// TIA Portal V18 export
FUNCTION "Room2_Main" : Void   // FC5, LAD
{ S7_Optimized_Access := 'TRUE' }
VERSION : 0.1
// stored: AutoNumber true, IsIECCheckEnabled false, SetENOAutomatically false, UDAEnableTagReadback false
BEGIN

REGION Network 1: 区域搜索
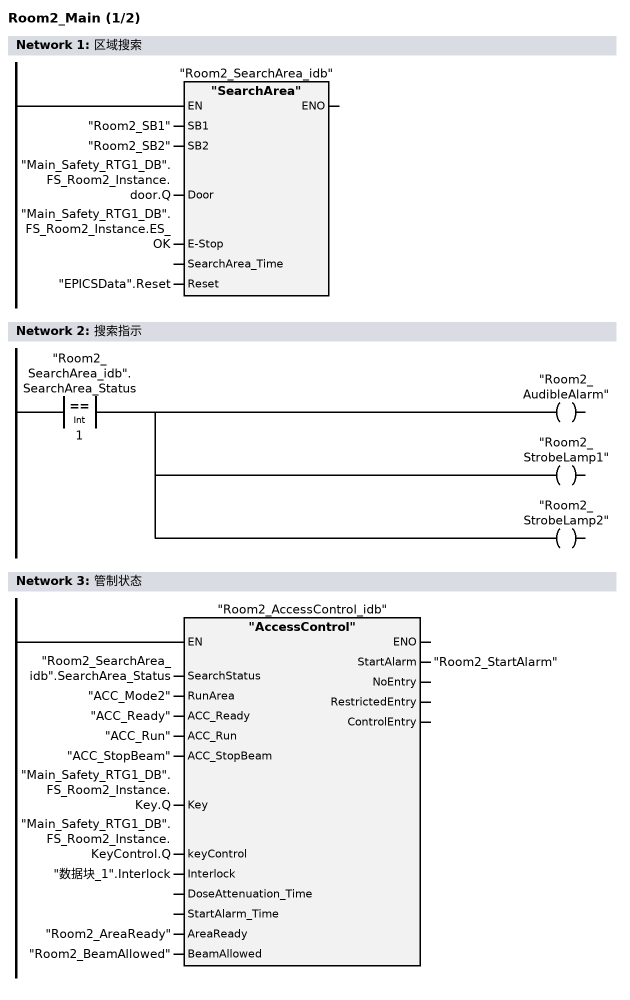
   RUNG wire#powerrail
      "Room2_SearchArea_idb"(SB1 := "Room2_SB1", SB2 := "Room2_SB2", Door := "Main_Safety_RTG1_DB".FS_Room2_Instance.door.Q, "E-Stop" := "Main_Safety_RTG1_DB".FS_Room2_Instance.ES_OK, SearchArea_Time :=, Reset := "EPICSData".Reset)
   END_RUNG
   // the same network as SCL:
   "Room2_SearchArea_idb"(SB1 := "Room2_SB1",   // "SearchArea"
                          SB2 := "Room2_SB2",
                          Door := "Main_Safety_RTG1_DB".FS_Room2_Instance.door.Q,
                          "E-Stop" := "Main_Safety_RTG1_DB".FS_Room2_Instance.ES_OK,
                          Reset := "EPICSData".Reset);
END_REGION

REGION Network 2: 搜索指示
   RUNG wire#powerrail
      { S7_Templates := "SrcType := Int" } EQ_Contact(in1 := "Room2_SearchArea_idb".SearchArea_Status, in2 := 1)
      wire#w1
      Coil( "Room2_AudibleAlarm" )
   END_RUNG
   RUNG wire#w1
      Coil( "Room2_StrobeLamp1" )
   END_RUNG
   RUNG wire#w1
      Coil( "Room2_StrobeLamp2" )
   END_RUNG
   // the same network as SCL:
   "Room2_AudibleAlarm" := "Room2_SearchArea_idb".SearchArea_Status = 1;
   "Room2_StrobeLamp1" := "Room2_AudibleAlarm";
   "Room2_StrobeLamp2" := "Room2_AudibleAlarm";
END_REGION

REGION Network 3: 管制状态
   RUNG wire#powerrail
      "Room2_AccessControl_idb"(SearchStatus := "Room2_SearchArea_idb".SearchArea_Status, RunArea := "ACC_Mode2", ACC_Ready := "ACC_Ready", ACC_Run := "ACC_Run", ACC_StopBeam := "ACC_StopBeam", Key := "Main_Safety_RTG1_DB".FS_Room2_Instance.Key.Q, keyControl := "Main_Safety_RTG1_DB".FS_Room2_Instance.KeyControl.Q, Interlock := "数据块_1".Interlock, DoseAttenuation_Time :=, StartAlarm_Time :=, AreaReady := "Room2_AreaReady", BeamAllowed := "Room2_BeamAllowed", StartAlarm => "Room2_StartAlarm", NoEntry =>, RestrictedEntry =>, ControlEntry =>)
   END_RUNG
   // the same network as SCL:
   "Room2_AccessControl_idb"(SearchStatus := "Room2_SearchArea_idb".SearchArea_Status,   // "AccessControl"
                           RunArea := "ACC_Mode2",
                           ACC_Ready := "ACC_Ready",
                           ACC_Run := "ACC_Run",
                           ACC_StopBeam := "ACC_StopBeam",
                           Key := "Main_Safety_RTG1_DB".FS_Room2_Instance.Key.Q,
                           keyControl := "Main_Safety_RTG1_DB".FS_Room2_Instance.KeyControl.Q,
                           Interlock := "数据块_1".Interlock,
                           AreaReady := "Room2_AreaReady",
                           BeamAllowed := "Room2_BeamAllowed",
                           StartAlarm => "Room2_StartAlarm");
END_REGION

REGION Network 4: 管制输出
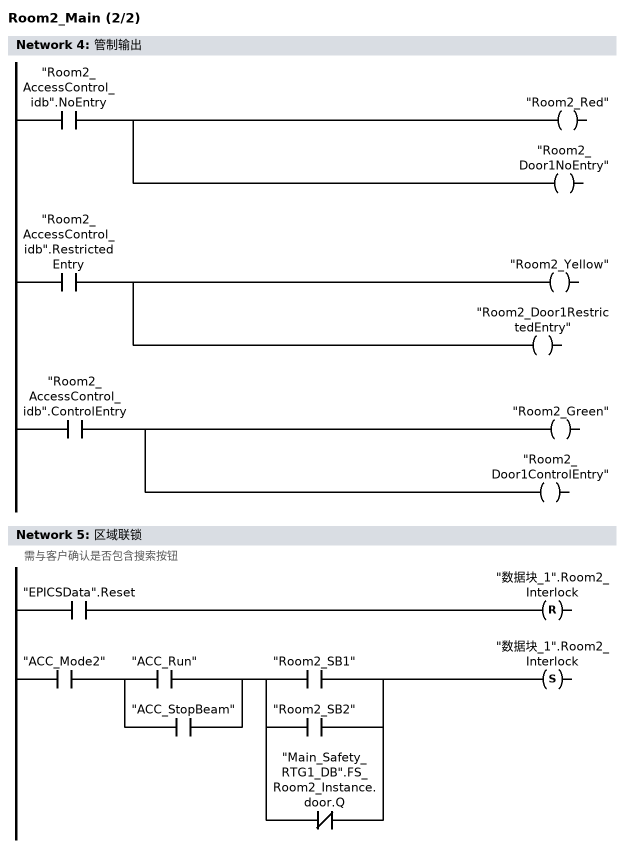
   RUNG wire#powerrail
      Contact( "Room2_AccessControl_idb".NoEntry )
      wire#w1
      Coil( "Room2_Red" )
   END_RUNG
   RUNG wire#w1
      Coil( "Room2_Door1NoEntry" )
   END_RUNG
   RUNG wire#powerrail
      Contact( "Room2_AccessControl_idb".RestrictedEntry )
      wire#w2
      Coil( "Room2_Yellow" )
   END_RUNG
   RUNG wire#w2
      Coil( "Room2_Door1RestrictedEntry" )
   END_RUNG
   RUNG wire#powerrail
      Contact( "Room2_AccessControl_idb".ControlEntry )
      wire#w3
      Coil( "Room2_Green" )
   END_RUNG
   RUNG wire#w3
      Coil( "Room2_Door1ControlEntry" )
   END_RUNG
   // the same network as SCL:
   "Room2_Red" := "Room2_AccessControl_idb".NoEntry;
   "Room2_Door1NoEntry" := "Room2_AccessControl_idb".NoEntry;
   "Room2_Yellow" := "Room2_AccessControl_idb".RestrictedEntry;
   "Room2_Door1RestrictedEntry" := "Room2_AccessControl_idb".RestrictedEntry;
   "Room2_Green" := "Room2_AccessControl_idb".ControlEntry;
   "Room2_Door1ControlEntry" := "Room2_AccessControl_idb".ControlEntry;
END_REGION

REGION Network 5: 区域联锁
   // 需与客户确认是否包含搜索按钮
   RUNG wire#powerrail
      Contact( "EPICSData".Reset )
      R_Coil( "数据块_1".Room2_Interlock )
   END_RUNG
   RUNG wire#powerrail
      Contact( "ACC_Mode2" )
      wire#w1
      Contact( "ACC_Run" )
      wire#w2
      Contact( "Room2_SB1" )
      wire#w3
      S_Coil( "数据块_1".Room2_Interlock )
   END_RUNG
   RUNG wire#w1
      Contact( "ACC_StopBeam" )
   END_RUNG wire#w2
   RUNG wire#w2
      Contact( "Room2_SB2" )
   END_RUNG wire#w3
   RUNG wire#w2
      I_Contact( "Main_Safety_RTG1_DB".FS_Room2_Instance.door.Q )
   END_RUNG wire#w3
   // the same network as SCL:
   IF "EPICSData".Reset THEN "数据块_1".Room2_Interlock := FALSE; END_IF;
   IF "ACC_Mode2" AND ("ACC_Run" OR "ACC_StopBeam") AND ("Room2_SB1" OR "Room2_SB2" OR NOT "Main_Safety_RTG1_DB".FS_Room2_Instance.door.Q) THEN
       "数据块_1".Room2_Interlock := TRUE;
   END_IF;
END_REGION
END_FUNCTION
